(* Schneider Machine Expert - Basic project New project, file version 2.4.0.0 *)
(* ProjectInformations: Name=New project *)

HARDWARE
  Cpu 0: TM221ME16R/G
  EthernetConfiguration: NetworkName=M221, IpAllocationMode=FixedAddress, IpAddress=0.0.0.0, SubnetMask=0.0.0.0
  SerialLineConfiguration: Baud=Baud19200, Parity=ParityEven, DataBits=DataBits8, StopBits=StopBits1, PhysicalMedium=PhysicalMediumRs485, TransmissionMode=TransmissionModeModbusRtu, SlaveId=1, Addressing=SlaveAddressing
  MastTask: UsePeriodScanMode=false, PeriodScan=100
  FastTask: Period=255
  CpuBehavior: StartingMode=StartAsPreviousState, AutoSaveRamOnEeprom=true, WatchdogPeriod=250

SYMBOLS  (address, symbol, comment, settings)
  %M0         "Транспортер1"
  %M1         "Датчик Д1"
  %M2         "Транспортер2"
  %M3         "Транспортер3"
  %M4         "Датчик2"
  %TM0        [Preset=3, Base=OneSecond]
  %TM1        [Preset=3, Base=OneSecond]
  %TM2        "Таймер выключения через 5 сек"  [Type=TOF, Preset=5, Base=OneSecond]

POU New POU
  (* SectionNumber=1 *)

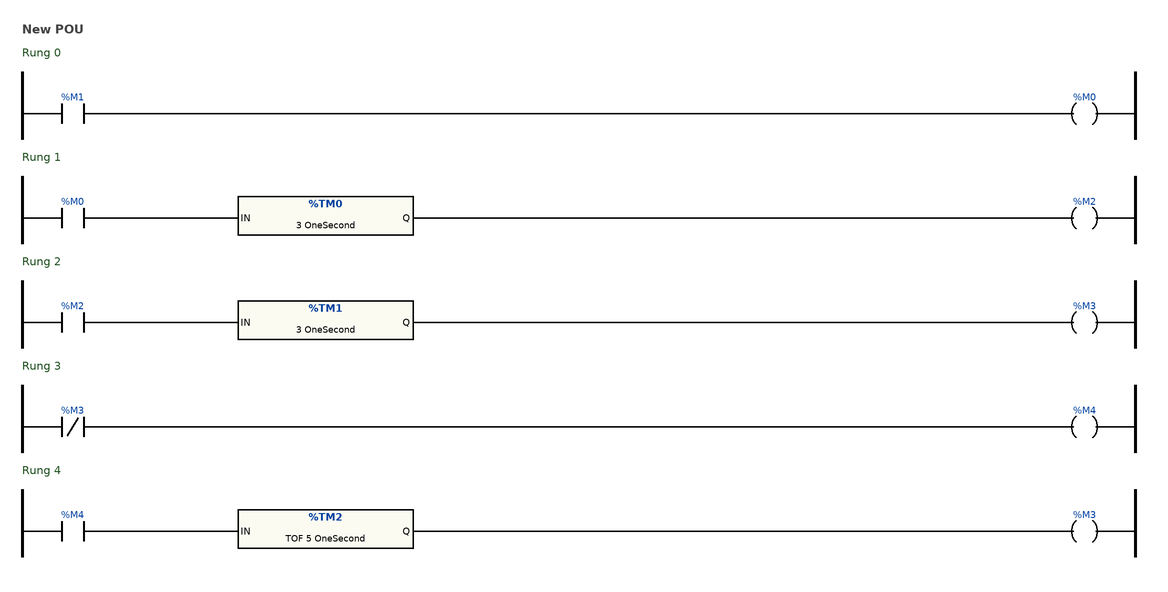

// Rung 0
  LD %M1
  ST %M0
  // as ST:
  //   %M0 := %M1;

// Rung 1
  BLK %TM0
  LD %M0
  IN
  OUT_BLK
  LD Q
  ST %M2
  END_BLK
  // as ST:
  //   %TM0(IN := %M0);
  //   %M2 := %TM0.Q;

// Rung 2
  BLK %TM1
  LD %M2
  IN
  OUT_BLK
  LD Q
  ST %M3
  END_BLK
  // as ST:
  //   %TM1(IN := %M2);
  //   %M3 := %TM1.Q;

// Rung 3
  LDN %M3
  ST %M4
  // as ST:
  //   %M4 := NOT %M3;

// Rung 4
  BLK %TM2
  LD %M4
  IN
  OUT_BLK
  LD Q
  ST %M3
  END_BLK
  // as ST:
  //   %TM2(IN := %M4);
  //   %M3 := %TM2.Q;
